FUNCTION_BLOCK fbPiston EXTENDS TcoCore.TcoComponent
VAR_INPUT
	iHomePositionSensor : BOOL;
	iWorkPositionSensor : BOOL;	
END_VAR

VAR_OUTPUT
	qHomePositionActuator : BOOL;
	qWorkPositionActuator : BOOL;		
END_VAR

VAR
	_moveHomeTask : fbPistonMoveTask(THIS^);
	_moveWorkTask : fbPistonMoveTask(THIS^);
END_VAR

_moveHomeTask(PositionSensor := iHomePositionSensor, MoveToPositionSignal := qHomePositionActuator, InverseSignal := qWorkPositionActuator);
_moveWorkTask(PositionSensor := iWorkPositionSensor, MoveToPositionSignal := qWorkPositionActuator, InverseSignal := qHomePositionActuator);

METHOD PROTECTED Manual
VAR_INPUT
END_VAR
END_METHOD

METHOD MoveHome : TcoCore.ITcoTask
MoveHome := THIS^._moveHomeTask.Invoke();
END_METHOD

METHOD MoveWork : TcoCore.ITcoTask
MoveWork := THIS^._moveWorkTask.Invoke();
END_METHOD

METHOD  Restore : ITcoRestorable
THIS^._moveHomeTask.Restore();
THIS^._moveWorkTask.Restore();
END_METHOD

END_FUNCTION_BLOCK

(* stored: Version 1.1.0.1, ProductVersion 3.1.4024.6
   POU fbPiston: Id {df7086e3-24fe-4034-ba31-b05bb5ffe13c}, SpecialFunc None
   Method Manual: Id {07a3a813-6109-4bbf-8965-f34f5d38a661}
   Method MoveHome: Id {4e7fadb5-1a48-4a7b-80f7-ff4252ecf17a}
   Method MoveWork: Id {5fe891ea-5923-4779-be52-a85d819af426}
   Method Restore: Id {b6ea9502-7703-4515-a330-5f9f26abdfef} *)
